TYPE ST_MasterCTRL :
STRUCT
	

	// Request Flags
	bHoming_Request						:BOOL;
	bProccess_Request					:BOOL;
	bStop_Request						:BOOL;
	bAbortAction_Request				:BOOL;
	bManualModeRequest					:BOOL;
	
	bCycleStopRequest					:BOOL;		
	bAllActionsStopped					:BOOL;
	bCycleStopFault						:BOOL;
	bNoMachineImmediateFault			:BOOL;
	bNoCycleStopFault					:BOOL;	
	bAllModulesReady					:BOOL;

	// Feedback Flags
	bAllModules_Homed					:BOOL;
	bAllModules_Stopped					:BOOL;
	bAllModules_Aborted					:BOOL;
	bPowerUpTimerComplete				:BOOL;

	
//-------------------------------------------------------------------------------oldschoo1
		
END_STRUCT
END_TYPE

(* stored: Version 1.1.0.1, ProductVersion 3.1.4024.12
   DUT ST_MasterCTRL: Id {0cf524b1-b3b8-486a-882b-6a9427e24a47} *)
